FUNCTION_BLOCK FB_Axis_NoHoming EXTENDS FB_AxisBase
VAR_INPUT
END_VAR
VAR_OUTPUT
END_VAR
VAR
END_VAR

METHOD MotionControl : BOOL
VAR_INPUT
END_VAR
SUPER^.MotionControl();

IF bDriveEnabled AND NOT SelectedAxis.Status.Homed THEN
	//Since homing does not matter for this axis, just home it wherever it sits when enabled
	fbAxisHome(
				Axis:= SelectedAxis, 
				Execute:= TRUE, 
				Position:= 0, 
				HomingMode:= MC_Direct, 
				BufferMode:= , 
				Options:= , 
				bCalibrationCam:= TRUE, 
				Done=> , 
				Busy=> , 
				Active=> , 
				CommandAborted=> , 
				Error=> , 
				ErrorID=> );
END_IF
END_METHOD

END_FUNCTION_BLOCK

(* stored: Version 1.1.0.1, ProductVersion 3.1.4024.9
   POU FB_Axis_NoHoming: Id {67f12062-5bd4-44d4-b963-30cd41ea59ee}, SpecialFunc None
   Folder 01_SUPER_Overrides: Id {cfe861f9-eb49-42ec-a7bf-5dfd11116946}
   Method MotionControl: Id {b0ccc3c6-e35f-4a18-adeb-ab31021524ff} *)
